FUNCTION Convert_LREAL_TO_TOD : Hresult
VAR_INPUT
	in : LREAL;
	out : REFERENCE TO TOD;
END_VAR
VAR
	converted : TOD;
END_VAR

converted := LREAL_TO_TOD(in);

IF (TOD_TO_LREAL(converted) <> in) THEN
	Convert_LREAL_TO_TOD := INCOMPATIBLE;
	RETURN;
END_IF

out := converted;

END_FUNCTION

(* stored: Version 1.1.0.1, ProductVersion 3.1.4024.12
   POU Convert_LREAL_TO_TOD: Id {7cbdf56f-335e-49ff-a81c-144fb07a746d}, SpecialFunc None *)
